(* PLC project Unnamed, Unknown Unnamed 1 *)
(* stored: creationDateTime 2023-12-01T09:12:27, modificationDateTime 2023-12-01T09:12:27 *)

CONFIGURATION Config0
  RESOURCE Res0 ON PLC
  END_RESOURCE
END_CONFIGURATION
